(* CODESYS project Controle de Nivel.project

Project tree, tasks and I/O mapping:
  Device : CODESYS Control Win V3, 3S - Smart Software Solutions GmbH, order no. 305021, version 3.5.11.30
    application Application
      libraries: Standard, * (System)
      task MainTask (cyclic, interval t#20ms, priority 1) calls PLC_PRG
      task VISU_TASK (cyclic, interval 100 ms, priority 31) calls VisuElems.Visu_Prg
      program PLC_PRG [LD]
      visualisation Visualization
      Symbols
  libraries: VisuSymbols, 3.5.10.0 (System)
  text list GlobalTextList
*)

// Device/Application/PLC_PRG
PROGRAM PLC_PRG
VAR
	NIVEL: REAL;
	SENSOR: REAL;
	V1: BOOL;
	B1: BOOL;
	V2: BOOL;
	AB0: BYTE;
END_VAR
VAR // added by the converter: edge detectors and wires of the graphical bodies
    _w1, _w2 : BOOL;
END_VAR

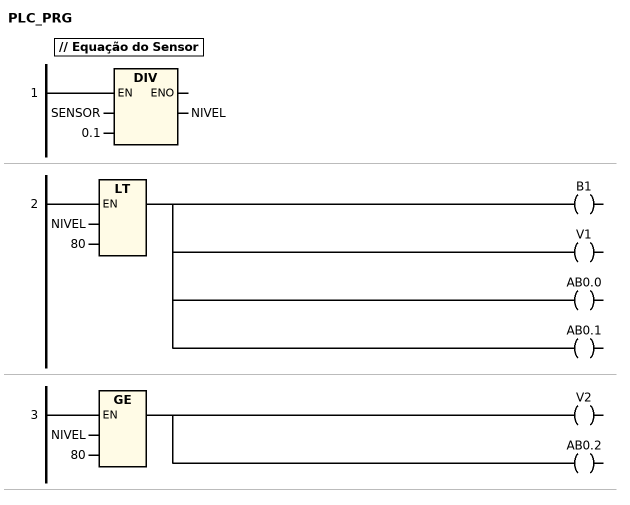
// NETWORK 1
// label: // Equação do Sensor
NIVEL := SENSOR / 0.1;

// NETWORK 2
_w1 := NIVEL < 80;
B1 := _w1;
V1 := _w1;
AB0.0 := _w1;
AB0.1 := _w1;

// NETWORK 3
_w2 := NIVEL >= 80;
V2 := _w2;
AB0.2 := _w2;

END_PROGRAM

// Device/Application/Visualization
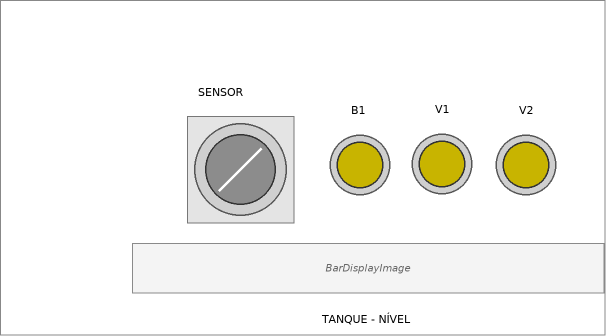
VISUALIZATION Visualization  // 606x336
    Potentiometer360 (168,116 145x107), variable: PLC_PRG.SENSOR, style: Potentiometer-Potentiometer360-Gray, scale format: %.1f, scale 0..10
        p2431819421: Outside
    BarDisplayImage (132,243 472x50), value: PLC_PRG.NIVEL, style: BarDisplayImage-Gray, scale format: %.1f, scale 0..100
    Lamp1 (325,130 70x70), variable: PLC_PRG.B1, style: Lamp-Lamp1-Yellow
    Lamp1 (407,129 70x70), variable: PLC_PRG.V1, style: Lamp-Lamp1-Yellow
    Label (335,96 47x29), "B1"
    Label (419,95 47x29), "V1"
    Label (171,78 99x29), "SENSOR"
    Label (267,305 198x29), "TANQUE - NÍVEL"
    Lamp1 (491,130 70x70), variable: PLC_PRG.V2, style: Lamp-Lamp1-Yellow
    Label (503,96 47x29), "V2"
END_VISUALIZATION
